// TwinCAT 3 PLC project PlcPresentationExamples
// ProgramVersion: 3.1.4023.0
// libraries:
//   Tc2_Standard, * (Beckhoff Automation GmbH)
//   Tc2_System, * (Beckhoff Automation GmbH)
//   Tc3_Module, * (Beckhoff Automation GmbH)
//   VortexBase, 0.101.0.30 (Vortex.Library)
// project tree:
//   / PlcTask.TcTTO
//   POUs/Counter/ stCounter.TcDUT
//   POUs/Enums/ enumMonths.TcDUT
//   POUs/ MAIN.TcPOU
//   POUs/Stations/01/ fbStation01.TcPOU, stStation01_Components.TcDUT, stStation01_Data.TcDUT
//   POUs/Stations/02/ fbStation02.TcPOU, stStation02_Components.TcDUT, stStation02_Data.TcDUT
//   POUs/Stations/ fbStations.TcPOU

CONFIGURATION PlcPresentationExamples
    RESOURCE PLC ON TwinCAT3
        TASK PlcTask(INTERVAL := T#10ms, PRIORITY := 21);
        PROGRAM MAIN WITH PlcTask : MAIN;
    END_RESOURCE
END_CONFIGURATION

// ---- POUs/Counter/stCounter.TcDUT
{attribute wpf [Container(Layout.Stack)]}
TYPE stCounter :
STRUCT
	{attribute addProperty Name "Allow counting"}
	{attribute addProperty ToolTip "Allows the counter to increment value."}
	_doCount : BOOL;
	{attribute addProperty Name "Counter"}
	{attribute addProperty ToolTip "Counter value."}
	_counterValue : INT;	
	{attribute addProperty Name "Reset Counter"}
	{attribute addProperty ToolTip "Resets counter to 0"}
	_resetCounterValue : BOOL;
END_STRUCT
END_TYPE

// ---- POUs/Enums/enumMonths.TcDUT
{attribute 'qualified_only'}
{attribute 'strict'}
TYPE enumMonths :
(
	January := 1,
	February := 2,
	March := 3,
	April := 4,
	May := 5,
	June := 6,
	July := 7,
	August := 8,
	September := 9,
	October := 10,
	November := 11,
	December := 12
);
END_TYPE

// ---- POUs/Stations/01/stStation01_Components.TcDUT
{attribute wpf [Container(Layout.Stack)]}
TYPE stStation01_Components :
STRUCT
	{attribute addProperty Name "Sensor X"}
	SensorX : REAL;
	
	{attribute wpf [Container(Layout.Wrap)]}
	{attribute addProperty Name "Upper piston sensor"}
	PistonUpPosition AT %I* : BOOL;
	{attribute addProperty Name "Bottom piston sensor"}
	PistonDownPosition AT %I* : BOOL;
	
	{attribute wpf [Container(Layout.Wrap)]}
	{attribute addProperty Name "Move up piston singal"}
	MovePistonUp AT %Q* : BOOL;
	{attribute addProperty Name "Move down piston singal"}
	MovePistonDown AT %Q* : BOOL;
END_STRUCT
END_TYPE

// ---- POUs/Stations/01/stStation01_Data.TcDUT
{attribute wpf [Container(Layout.Stack)]}
TYPE stStation01_Data :
STRUCT
	{attribute addProperty Name "X Min"}
	DimXMin : REAL;	
	{attribute clr [ReadOnly()]}
	{attribute addProperty Name "X Measured"}
	DimXMeasured : REAL;	
	{attribute addProperty Name "X Max"}
	DimXMax : REAL;
	{attribute addProperty Name "Result"}
	Result : STRING;
END_STRUCT
END_TYPE

// ---- POUs/Stations/02/stStation02_Components.TcDUT
{attribute wpf [Container(Layout.Stack)]}
TYPE stStation02_Components :
STRUCT
	{attribute addProperty Name "Sensor Y"}
	SensorY : REAL;
END_STRUCT
END_TYPE

// ---- POUs/Stations/02/stStation02_Data.TcDUT
{attribute wpf [Container(Layout.Stack)]}
TYPE stStation02_Data :
STRUCT
	{attribute wpf [Container(Layout.Wrap)]}
	{attribute addProperty Name "Y Min"}
	DimYMin : REAL;
	{attribute addProperty Name "Y Measured"}
	DimYMeasured : REAL;
	{attribute addProperty Name "Y Max"}
	DimYMax : REAL;
	{attribute addProperty Name "Result"}
	
	{attribute wpf [Container(Layout.Stack)]}	
	Result : STRING;
END_STRUCT
END_TYPE

// ---- POUs/MAIN.TcPOU
{attribute wpf [Container(Layout.Tabs)]}
PROGRAM MAIN
VAR
	_counter : stCounter;
	_stations : fbStations;
	_months : enumMonths;
END_VAR

IF(_counter._doCount) THEN
	_counter._counterValue :=  _counter._counterValue + 1;
END_IF

IF(_counter._resetCounterValue) THEN
	_counter._counterValue := 0;
	_counter._resetCounterValue := FALSE;
END_IF

_stations();

END_PROGRAM

// ---- POUs/Stations/fbStations.TcPOU
{attribute wpf [Container(Layout.Tabs)]}
FUNCTION_BLOCK fbStations
VAR
	_st01 : fbStation01;
	_st02 : fbStation02;
END_VAR

_st01();
_st02();

END_FUNCTION_BLOCK

// ---- POUs/Stations/01/fbStation01.TcPOU
{attribute wpf [Container(Layout.Stack)]}
{attribute wpf [Group(Layout.Scroll)]}
{attribute addProperty Name "ST 01"}
FUNCTION_BLOCK fbStation01
VAR	
	{attribute wpf [Container(Layout.Wrap)]}
	{attribute addProperty Name "Step Number"}
	{attribute clr [ReadOnly()]}
	_step : INT;
	{attribute addProperty Name "Step description"}
	{attribute clr [ReadOnly()]}
	_stepDescription : STRING;
	{attribute wpf [Container(Layout.Wrap)]}	
	{attribute addProperty Name "Data"}
	_data : stStation01_Data;
	{attribute addProperty Name "Components"}
	_components : stStation01_Components;
END_VAR

CASE _step OF
	0:	_stepDescription := 'Moving piston down';
	
		_components.MovePistonDown := TRUE;
		_components.MovePistonUp := FALSE;
		
		IF(_components.PistonDownPosition) THEN
			_step := 10;
		END_IF
	10: _stepDescription := 'Taking measures';
		_data.DimXMeasured := _components.SensorX;
		IF(_data.DimXMin <= _data.DimXMeasured AND
			_data.DimXMeasured <= _data.DimXMax) THEN	
			_data.Result := 'ALL OK';
		ELSE
			_data.Result := 'THIS IS NOT OK';
		END_IF
		_step := 20;
	20: _stepDescription := 'Moving piston up';
		_components.MovePistonUp := TRUE;
		_components.MovePistonDown := FALSE;
		IF(_components.PistonUpPosition) THEN
			_step := 0;
		END_IF			
END_CASE

END_FUNCTION_BLOCK

// ---- POUs/Stations/02/fbStation02.TcPOU
{attribute wpf [Container(Layout.Tabs)]}
{attribute addProperty Name "ST 02"}
FUNCTION_BLOCK fbStation02
VAR
	{attribute wpf [Container(Layout.Stack)]}
	{attribute addProperty Name "Compare"}
	_compare : BOOL;
	{attribute addProperty Name "Data"}
	_data : stStation02_Data;
	{attribute addProperty Name "Components"}
	_components : stStation02_Components;
END_VAR

_data.DimYMeasured := _components.SensorY;
IF(_data.DimYMin <= _data.DimYMeasured AND
 	_data.DimYMeasured <= _data.DimYMax) THEN	
	_data.Result := 'ALL OK';
ELSE
	_data.Result := 'THIS IS NOT OK';
END_IF

END_FUNCTION_BLOCK
